FUNCTION_BLOCK INTERNAL FB_DummyObject EXTENDS FB_Object
VAR_INPUT
END_VAR
VAR_OUTPUT
END_VAR
VAR
    _nTest: INT;
END_VAR

PROPERTY nTest : INT
GET
nTest := THIS^._nTest;
END_GET
SET
THIS^._nTest := nTest;
END_SET
END_PROPERTY

END_FUNCTION_BLOCK

(* stored: Version 1.1.0.1, ProductVersion 3.1.4024.12
   POU FB_DummyObject: Id {02b827fa-a864-0b79-18d9-0983e456a88d}, SpecialFunc None
   Property nTest: Id {f39036c8-376b-0437-0832-34bdf02a2176}
   Get Get: Id {d8777a8d-ef56-00b5-16db-51fe57934994}
   Set Set: Id {aa98e316-bb19-0f2b-0301-2cc1ce295fbe} *)
